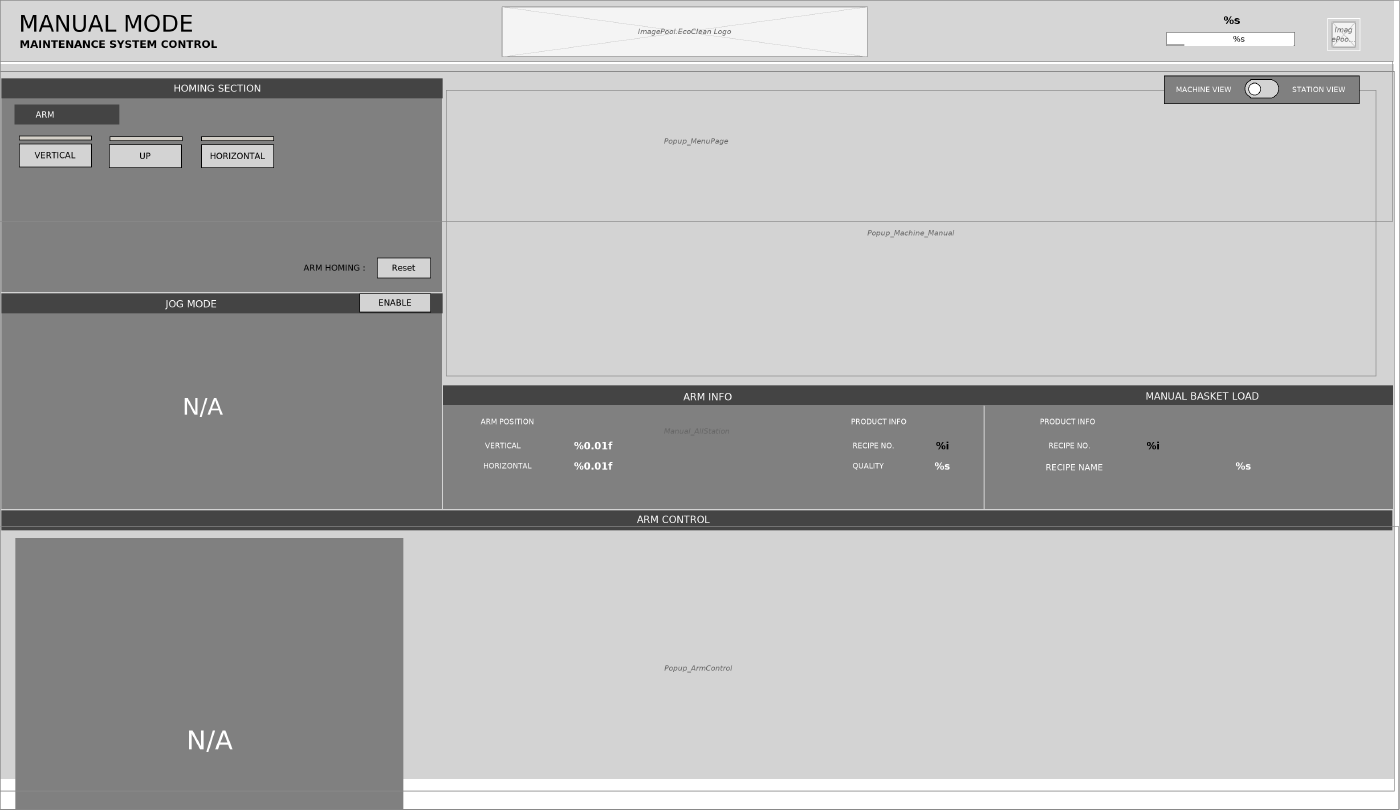
VISUALIZATION Manual_Page  // 1928x1116
    Rectangle (0,88 1919x985)
    Rectangle (1356,531 562x27)
    Rectangle (1356,558 562x143)
    Rectangle (2,431 606x270)
    Rectangle (2,135 606x267)
    Rectangle (2,703 1915x27)
    Rectangle (2,404 607x27)
    Rectangle (610,531 746x27)
    Rectangle (610,558 744x143)
    Rectangle (0,63 1920x26)
        p3528305787: HMI_Ctrl.ANIMATION3
    Rectangle (0,0 1919x85)
    Label (23,6 564x53), "MANUAL MODE"
    Label (24,49 541x24), "MAINTENANCE SYSTEM CONTROL"
    Group (1828,25 45x45)
        OnMouseClick: toggle HMI_Ctrl.MenuButton
        RoundedRectangle (0,0 45x45), colour toggle: HMI_Ctrl.MenuButton
        Image (6,5 33x35), image: ImagePool.Menu Button
    Frame (614,124 1281x394)
        shows Popup_Machine_Manual()
    Group (20,144 357x87)
        Group (0,0 144x27)
            Rectangle (0,0 144x27)
            Label (14,2 56x24), "ARM"
        Group (6,43 100x43)
            RoundedRectangle (0,0 100x6), colour toggle: ARbArmVertHomeDone[1]
            Rectangle (0,11 100x32), "VERTICAL", colour toggle: bArm1VertHomeStart_30
                toggle bArm1VertHomeStart_30
        Group (130,44 101x43)
            RoundedRectangle (1,0 100x6), colour toggle: ARDSArmCtrl[1].AR3sbPositionCfm[2,1,1]
            Rectangle (0,11 100x32), "UP", colour toggle: bArm1VertLD1Up_30
                toggle bArm1VertLD1Up_30
        Group (257,44 100x43)
            RoundedRectangle (0,0 100x6), colour toggle: ARbArmHorzHomeDone[1]
            Rectangle (0,11 100x32), "HORIZONTAL", colour toggle: bArm1HorzHomeStart_30
                toggle bArm1HorzHomeStart_30
    Group (405,355 188x28)
        Label (0,2 112x24), "ARM HOMING :"
        Rectangle (114,0 74x28), "Reset", colour toggle: bArmHomeResetbit
            tap bArmHomeResetbit
    Label (659,569 110x24), "ARM POSITION"
    Label (1169,569 110x24), "PRODUCT INFO"
    Label (1171,602 82x24), "RECIPE NO."
    Label (1171,630 63x24), "QUALITY"
    Rectangle (1248,606 100x17), "%i", text variable: DSArmBasketInfo[1].iProductRecipeNo
        OnMouseDown: write the text variable via VisuDialogs.Numpad, min 0, max 40
    Rectangle (1248,634 100x17), "%s", text variable: DSArmBasketInfo[1].sProductQuality
    Image (691,9 504x69), image: ImagePool.EcoClean Logo
    Frame (-2,725 1928x391)
        shows Popup_ArmControl()
    Label (856,704 143x24), "ARM CONTROL"
    Rectangle (742,634 150x17), "%0.01f", text variable: DSArm1HorzConfig.lrGen_Out_CurrentPos
    Label (638,602 82x24), "VERTICAL"
    Label (638,630 97x24), "HORIZONTAL"
    Rectangle (742,606 150x17), "%0.01f", text variable: DSArm1VertConfig.lrGen_Out_CurrentPos
    Label (908,535 133x24), "ARM INFO"
    Group (43,442 249x248)
        Ellipse (0,0 249x248)
        RoundedRectangle (90,12 70x223)
        RoundedRectangle (13,89 224x69)
        RoundedRectangle (89,88 73x72)
        Group (92,163 70x69)
            tap ARbArmVertJogFwd[1]
            PushSwitch (0,0 70x69), variable: ARbArmVertJogFwd[1], behaviour: TOGGLE, style: Switch-PushSwitch-Blue
            Image (14,17 40x40), image: VisuSymbols.Symbols.TriangleDown
        Group (17,89 70x69)
            tap ARbArmHorzJogRwd[1]
            PushSwitch (0,0 70x69), variable: ARbArmHorzJogRwd[1], behaviour: TOGGLE, style: Switch-PushSwitch-Blue
            Image (10,14 40x40), image: VisuSymbols.Symbols.TriangleLeft
        Group (165,89 70x69)
            tap ARbArmHorzJogFwd[1]
            PushSwitch (0,0 70x69), variable: ARbArmHorzJogFwd[1], behaviour: TOGGLE, style: Switch-PushSwitch-Blue
            Image (17,14 40x40), image: VisuSymbols.Symbols.TriangleRight
        Group (91,17 70x69)
            tap ARbArmVertJogRwd[1]
            PushSwitch (0,0 70x69), variable: ARbArmVertJogRwd[1], behaviour: TOGGLE, style: Switch-PushSwitch-Blue
            Image (15,11 40x40), image: VisuSymbols.Symbols.TriangleUp
    Rectangle (303,547 220x27)
    Label (329,550 157x24), "ARM JOG VELO (mm/s)"
    Label (310,587 82x24), "VERTICAL"
    Label (310,618 97x24), "HORIZONTAL"
    Rectangle (420,592 120x17), "%0.01f", text variable: ARrArmVertJogPercent[1]
        OnMouseDown: write the text variable via VisuDialogs.Numpad, min 2, max 100
    Rectangle (420,623 121x17), "%0.01f", text variable: ARrArmHorzJogPercent[1]
        OnMouseDown: write the text variable via VisuDialogs.Numpad, min 2, max 100
    Label (410,618 13x24), ":"
    Label (410,588 13x24), ":"
    Rectangle (2,108 607x27)
    Label (226,110 147x24), "HOMING SECTION"
    Label (215,407 97x24), "JOG MODE"
    Group (9,437 569x260), invisible if: bArmJogEnable
        Rectangle (0,0 525x255), invisible if: bArmJogEnable
        Label (184,94 173x59), "N/A", invisible if: bArmJogEnable
    Group (21,741 1876x333)
        Rectangle (0,0 534x610), invisible if: bArmHomingComplete[1]
        Label (199,194 138x170), "N/A", invisible if: bArmHomingComplete[1]
    Rectangle (495,404 98x26), "ENABLE", colour toggle: bArmJogEnable
        toggle bArmJogEnable
    Group (1603,103 269x41), invisible if: HMI_Ctrl.AutoStationViewEnable
        RoundedRectangle (0,1 269x39)
        Label (1,0 108x41), "MACHINE VIEW"
        Label (161,0 105x41), "STATION VIEW"
        Group (111,6 47x26)
            OnMouseClick: toggle HMI_Ctrl.AutoStationViewEnable
            Group (0,0 47x26)
                Ellipse (0,0 26x26)
                Ellipse (21,0 26x26)
                RoundedRectangle (8,0 29x26)
            Ellipse (1,1 24x24)
            Ellipse (23,1 23x24)
            RoundedRectangle (9,1 28x24)
            Ellipse (5,5 17x17)
    Group (1606,17 179x46)
        Button (0,27 177x19), image: VisuSymbols.Symbols.AddUser
        Rectangle (25,28 150x18), "%s", text variable: fbHmiTF1800_UserlevelManagement.dsHmiUserStatus_Active.sLoginName
        Rectangle (2,0 177x22), "%s", text variable: DSLocalSystemTimeML.sCurrentDT24Hr_General
    Label (1558,534 196x24), "MANUAL BASKET LOAD"
    Label (1437,632 127x24), "RECIPE NAME"
    Label (1429,569 110x24), "PRODUCT INFO"
    Label (1441,602 82x24), "RECIPE NO."
    Rectangle (1538,634 349x17), "%s", text variable: ARsProductRecipeDescription[iUserDefineProductRecipeNo]
    Rectangle (1538,606 100x17), "%i", text variable: iUserDefineProductRecipeNo
        OnMouseDown: write the text variable via VisuDialogs.Numpad, min 0, max 40
    Frame (0,98 1920x992), invisible if: NOT HMI_Ctrl.AutoStationViewEnable
        shows Manual_AllStation()
    Frame (0,84 1918x221), invisible if: HMI_Ctrl.CloseMenuButton
        shows Popup_MenuPage()
END_VISUALIZATION

(* stored: Version 1.1.0.1, ProductVersion 3.1.4024.12
   Visu Manual_Page: Id {29be1042-8c32-4274-a37f-12d573b92ca1} *)
